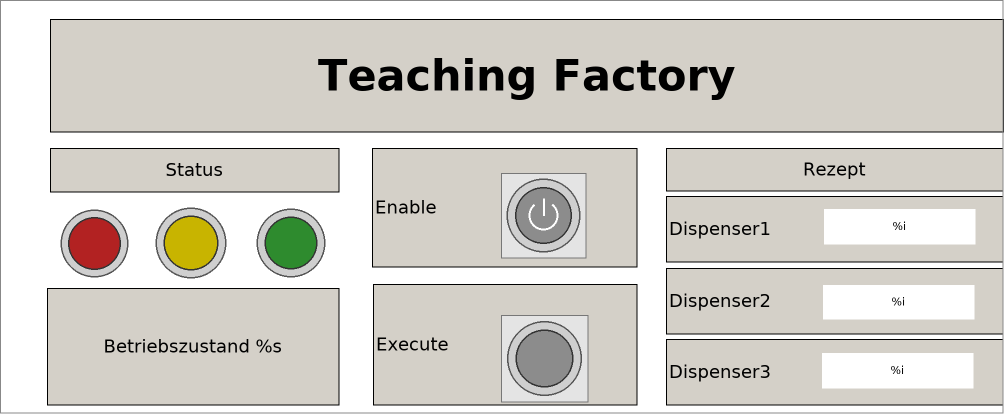
VISUALIZATION Visualization  // 1004x414
    Rectangle (666,196 337x66), "Dispenser1"
    Rectangle (50,19 954x113), "Teaching Factory"
    Lamp1 (55,202 79x83), variable: bAmpelRot, style: Lamp-Lamp1-Red
    Lamp1 (148,202 86x82), variable: bAmpelGelb, style: Lamp-Lamp1-Yellow
    Lamp1 (248,203 86x80), variable: bAmpelGrun, style: Lamp-Lamp1-Green
    Rectangle (50,148 289x44), "Status"
    Textfield (823,208 153x37), "%i", text variable: iBandFullmenge1
        p4168582468: iBandFullmenge1
        OnMouseDown: write the text variable via VisuDialogs.Numpad
    Rectangle (666,268 337x66), "Dispenser2"
    Rectangle (666,339 337x66), "Dispenser3"
    Rectangle (372,148 265x119), "Enable"
    Rectangle (373,284 264x121), "Execute"
    PowerSwitch (501,172 85x87), variable: bEnable, behaviour: TOGGLE, style: Switch-PowerSwitch-Gray
    PushSwitch (501,303 87x111), variable: bExecute, behaviour: TAP, style: Switch-PushSwitch-Gray
    Rectangle (666,148 337x43), "Rezept"
    Rectangle (47,288 292x117), "Betriebszustand %s", text variable: MAIN.fb_Ampelleuchte.eState
    Textfield (822,284 153x36), "%i", text variable: iBandFullmenge2
        p4168582468: iBandFullmenge2
        OnMouseDown: write the text variable via VisuDialogs.Numpad
    Textfield (821,352 153x37), "%i", text variable: iBandFullmenge3
        p4168582468: iBandFullmenge3
        OnMouseDown: write the text variable via VisuDialogs.Numpad
END_VISUALIZATION

(* stored: Version 1.1.0.1, ProductVersion 3.1.4024.15
   Visu Visualization: Id {845fa8cd-5b62-42da-a26b-aa21a88d7aeb} *)
